FUNCTION_BLOCK FB_TelescopeParkingState EXTENDS FB_TelescopeState
VAR_INPUT
END_VAR
VAR_OUTPUT
END_VAR
VAR
END_VAR

// 
// state
//

// run until parked
IF pMachine^.pControl^._Park() THEN
	pMachine^.State := E_TelescopeState.parked;
END_IF

END_FUNCTION_BLOCK

(* stored: Version 1.1.0.1, ProductVersion 3.1.4024.15
   POU FB_TelescopeParkingState: Id {8fc7bbd0-af57-48f4-8734-b825cd8fa56c}, SpecialFunc None *)
